(*
Geodetic Ellipsoid
----------------

Overview
================

Represents a geodetic reference ellipsoid (but not a geodetic datum). Contains functions for transitioning between latitude/longitude and XYZ coordinates.

To access standard ellipsoids use the GVL 'GeoEllipsoids'.	They cannot be copied, but you can use REFERENCE TO types to keep a shorthand copy somewhere.

.. note:: When creating an instance of this FB you *must* provide the name, semimajor axis, and flattening due to the use of FB_init parameters.
*)
{attribute 'no_assign'}
FUNCTION_BLOCK GeoEllipsoid
VAR_INPUT
END_VAR
VAR_OUTPUT
END_VAR
VAR
	Name_ : T_MaxString;
	SemiMajorAxis_ : LREAL;
	Flattening_ : LREAL;
END_VAR

METHOD FB_init : BOOL
VAR_INPUT
	bInitRetains : BOOL; // if TRUE, the retain variables are initialized (warm start / cold start)
	bInCopyCode : BOOL;  // if TRUE, the instance afterwards gets moved into the copy code (online change)
	
	eName : T_MaxString;
	eSemiMajorAxis : LREAL;//meters
	eFlattening : LREAL;//very small number
END_VAR
Name_ := eName;
SemiMajorAxis_ := eSemiMajorAxis;
Flattening_ := eFlattening;
END_METHOD

PROPERTY PUBLIC Flattening : LREAL
GET
Flattening := Flattening_;
END_GET
END_PROPERTY

METHOD PUBLIC GetCartesianFromGeodetic : Vector3
VAR_INPUT
	P : GeoPosition;
END_VAR
VAR
	N : LREAL;
END_VAR
N := GetNormalRadiusOfCurvature(P.LatitudeRad);

GetCartesianFromGeodetic.X := (N + P.Elevation) * COS(P.LatitudeRad) * COS(P.LongitudeRad);
GetCartesianFromGeodetic.Y := (N + P.Elevation) * COS(P.LatitudeRad) * SIN(P.LongitudeRad);
GetCartesianFromGeodetic.Z := ((1.0 - GetEccentricitySquared())*N + P.Elevation) * SIN(P.LatitudeRad);
END_METHOD

METHOD PROTECTED GetEccentricitySquared : LREAL
VAR_INPUT
END_VAR
GetEccentricitySquared := (2.0-Flattening)*Flattening;
END_METHOD

METHOD PROTECTED GetGeocentricLatitude : LREAL//radians
VAR_INPUT
	GeodeticLatitude : LREAL;//radians
END_VAR
GetGeocentricLatitude := ATAN((1-Flattening_) * (1-Flattening_)*TAN(GeodeticLatitude));
END_METHOD

METHOD PUBLIC GetGeodeticFromCartesian : GeoPosition
VAR_INPUT
	V : Vector3;
END_VAR
VAR
	RadLatitude_2 : LREAL;// 		'Q^2' 		from paper
	Magnitude_2 : LREAL;// 			'r^2' 		from paper
	Eccentricity_2 : LREAL;// 		'E^2' 		from paper
	AdjustedMag_2 : LREAL;// 		'r^2 - E^2' from paper
	SemiMinorConfocal_2 : LREAL;// 	'u^2' 		from paper
	SemiMajorConfocal_2 : LREAL;// 	'u^2' + E^2 from paper
	TanGeocentricLatitude : LREAL;// tan(beta) 	from paper
	GeocentricLatitude : LREAL;//   'beta' 		from paper
	AxialElevation : LREAL;
	RadialElevation : LREAL;
END_VAR
//stolen from : http://ir.lib.ncku.edu.tw/bitstream/987654321/39750/1/3011200501001.pdf
//error is <1mm for anything within 100km of the surface of the earth

RadLatitude_2 := V.X*V.X + V.Y*V.Y;
Magnitude_2 := RadLatitude_2 + V.Z* V.Z;

//right at pole longitude is indetermiante
IF RadLatitude_2 = 0 THEN
	GetGeodeticFromCartesian.LongitudeRad := 0;
ELSE
	GetGeodeticFromCartesian.LongitudeRad := atan2(V.Y,V.X);//eq 4c from paper
END_IF

//too close to poles for stuff to work well
IF RadLatitude_2 < (SemiMajorAxis * SemiMinorAxis * 1E-32) THEN
	//center of earth...angles dont even matter anymore
	IF V.Z = 0 THEN
		GetGeodeticFromCartesian.LatitudeRad := 0;
		GetGeodeticFromCartesian.Elevation := Magnitude_2;
	ELSE
		GetGeodeticFromCartesian.LatitudeRad := PI /2 * V.Z / ABS(V.Z);
		GetGeodeticFromCartesian.Elevation := ABS(V.Z) - SemiMinorAxis;
	END_IF;
ELSE
	Eccentricity_2 := SemiMajorAxis*SemiMajorAxis - SemiMinorAxis * SemiMinorAxis;
	AdjustedMag_2 := Magnitude_2 - Eccentricity_2;
	SemiMinorConfocal_2 := 0.5*AdjustedMag_2 + 0.5*SQRT(EXPT(AdjustedMag_2,2) + 4*Eccentricity_2*V.Z*V.Z); //eq 4a from paper
	SemiMajorConfocal_2 := SemiMinorConfocal_2 + Eccentricity_2;
	IF SQRT(SemiMinorConfocal_2) / SQRT(SemiMajorConfocal_2) < 10E-10 THEN
		//avoid divide by near zero when confocal is nearly flat and assumption of geocentric latidude equivalence atan(confocal) ~= atan(ellipsoid) stops being true
		IF V.Z = 0 THEN
			GeocentricLatitude := 0;
		ELSE
			GeocentricLatitude := PI/2 * V.Z/ABS(V.Z);
		END_IF;
		GetGeodeticFromCartesian.LatitudeRad := GeocentricLatitude;
	ELSE
		TanGeocentricLatitude := (SQRT(SemiMajorConfocal_2) * V.Z) / (SQRT(SemiMinorConfocal_2)*SQRT(RadLatitude_2));
		GeocentricLatitude := ATAN(TanGeocentricLatitude); //eq 6 from paper
		GetGeodeticFromCartesian.LatitudeRad := ATAN(SemiMajorAxis / SemiMinorAxis * TanGeocentricLatitude);
	END_IF;
	
	AxialElevation := V.Z - SemiMinorAxis*SIN(GeocentricLatitude);
	RadialElevation := SQRT(RadLatitude_2) - SemiMajorAxis*COS(GeocentricLatitude);
	
	GetGeodeticFromCartesian.Elevation := SQRT(AxialElevation*AxialElevation + RadialElevation*RadialElevation); //eq 7 from paper
	IF AxialElevation < 0 AND RadialElevation < 0 THEN
		GetGeodeticFromCartesian.Elevation := -1 * GetGeodeticFromCartesian.Elevation;
	END_IF

END_IF
END_METHOD

METHOD PROTECTED GetNormalRadiusOfCurvature : LREAL
VAR_INPUT
	lat : LREAL;//radians
END_VAR
VAR
	acosf : LREAL;
	bcosf : LREAL;
	den : LREAL;
END_VAR
acosf := SemiMajorAxis * COS(lat);
bcosf := GetSemiMinorAxis() * SIN(lat);
den := SQRT(acosf*acosf + bcosf*bcosf);
IF den = 0 THEN
	GetNormalRadiusOfCurvature := 0;
	ADSLOGSTR(ADSLOG_MSGTYPE_WARN,'GeodeticPosition::GetNormalRadiusOfCurvature Divide By Zero attempt in reference ellipsoid %s',Name);
	RETURN;
END_IF
GetNormalRadiusOfCurvature := SemiMajorAxis*SemiMajorAxis/den;
END_METHOD

METHOD PROTECTED GetSemiMinorAxis : LREAL
VAR_INPUT
END_VAR
GetSemiMinorAxis := SemiMajorAxis * (1-Flattening);
END_METHOD

METHOD PUBLIC GetTangentEnuRotation : RMatrix
VAR_INPUT
	P : GeoPosition;
END_VAR
VAR
	R_ENU : RMatrix;
	R_Lon : Rmatrix;
	R_Lat : Rmatrix;
	V : Vector3;
END_VAR
GetTangentEnuRotation := GetTangentXyuRotation(P,0.0);
RETURN;

//ECEF has X as 'up',   y as 'east',  Z as 'north' as lat=lon=0, translated to surface
//ENU  has X as 'east', y as 'north', z as 'up'
//therefore, the base rotation (ignoring lat/lon changes) should be: (projecting ENU unit vecotrs onto ECEF CS)
// [  0   0   1
//    1   0   0
//    0   1   0   ]

GetTangentEnuRotation.FillTrapezoidal(0,0,0);
GetTangentEnuRotation.SetRC(1,0,1);
GetTangentEnuRotation.SetRC(2,1,1);
GetTangentEnuRotation.SetRC(0,2,1);


R_Lon.SetFromAngle(P.LongitudeRad,Dimension.Z);//positive intrinsic rotation around ECEF Z
R_Lat.SetFromAngle(-1*P.LatitudeRad,Dimension.Y);//negative instrinsic rotation around rotated ECEF Y

GetTangentEnuRotation.RotateBy(R_Lat);
GetTangentEnuRotation.RotateBy(R_Lon);
END_METHOD

METHOD PUBLIC GetTangentEnuTransform : HMatrix
VAR_INPUT
	P : GeoPosition;
END_VAR
VAR
	R_ENU : RMatrix;
	R_Lon : Rmatrix;
	R_Lat : Rmatrix;
	V : Vector3;
END_VAR
V := GetCartesianFromGeodetic(P);
GetTangentEnuTransform.SetFromComponents(GetTangentEnuRotation(P),V);
END_METHOD

METHOD PUBLIC GetTangentXyuRotation : RMatrix
VAR_INPUT
	P : GeoPosition;
	Angle : LREAL;//radians of extra angle around the 'up' vector, from ENU
END_VAR
VAR
	R_ENU : RMatrix;
	R_Lon : Rmatrix;
	R_Lat : Rmatrix;
	RHeading : RMatrix;
	V : Vector3;
END_VAR
//ECEF has X as 'up',   y as 'east',  Z as 'north' as lat=lon=0, translated to surface
//ENU  has X as 'east', y as 'north', z as 'up'
//therefore, the base rotation (ignoring lat/lon changes) should be: (projecting ENU unit vecotrs onto ECEF CS)
// [  0   0   1
//    1   0   0
//    0   1   0   ]

GetTangentXyuRotation.SetFromAngle(Angle,Dimension.Z);

R_ENU.FillTrapezoidal(0,0,0);
R_ENU.SetRC(1,0,1);
R_ENU.SetRC(2,1,1);
R_ENU.SetRC(0,2,1);

R_Lon.SetFromAngle(P.LongitudeRad,Dimension.Z);//positive intrinsic rotation around ECEF Z
R_Lat.SetFromAngle(-1*P.LatitudeRad,Dimension.Y);//negative instrinsic rotation around rotated ECEF Y

GetTangentXyuRotation.RotateBy(R_ENU);
GetTangentXyuRotation.RotateBy(R_Lat);
GetTangentXyuRotation.RotateBy(R_Lon);
END_METHOD

METHOD PUBLIC GetTangentXyuTransform : HMatrix
VAR_INPUT
	P : GeoPosition;
	Angle : LREAL;//radians of extra normal rotation
END_VAR
VAR
	R_ENU : RMatrix;
	R_Lon : Rmatrix;
	R_Lat : Rmatrix;
	V : Vector3;
END_VAR
V := GetCartesianFromGeodetic(P);
GetTangentXyuTransform.SetFromComponents(GetTangentXyuRotation(P,Angle),V);
END_METHOD

PROPERTY PUBLIC Name : T_MaxString
GET
Name := Name_;
END_GET
END_PROPERTY

//meters
PROPERTY PUBLIC SemiMajorAxis : LREAL
GET
SemiMajorAxis := SemiMajorAxis_;
END_GET
END_PROPERTY

PROPERTY PUBLIC SemiMinorAxis : LREAL
GET
SemiMinorAxis := SemiMajorAxis*(1-Flattening);
END_GET
END_PROPERTY

END_FUNCTION_BLOCK

(* stored: Version 1.1.0.1, ProductVersion 3.1.4024.9
   POU GeoEllipsoid: Id {5fa9ec91-c8df-4619-93de-f428fe8da353}, SpecialFunc None
   Folder Helpers: Id {b81f80d4-2bbb-4268-8ddd-c7326c54d401}
   Folder Properties: Id {b4f92432-ea7a-4ff4-815d-4808dee4ca34}
   Folder Protected: Id {d95a2200-fe2b-4706-b87d-15a39d09296c}
   Method FB_init: Id {356473b9-f5c8-4741-9e86-0658e3600f83}
   Property Flattening: Id {34b2fe7f-e49d-4b2c-8e6e-38d008c42ac1}
   Get Get: Id {5861998b-a1c7-428b-b4da-036da0771533}
   Method GetCartesianFromGeodetic: Id {3dee90e0-402c-4ec5-8ec8-6eb06ee928ca}
   Method GetEccentricitySquared: Id {dcf07e5e-00c3-480f-9648-fb9fcd18870b}
   Method GetGeocentricLatitude: Id {7fa6146d-71cd-4c31-88c4-e5b241b37441}
   Method GetGeodeticFromCartesian: Id {9f899f33-9489-4cc0-a19d-4c589c0cda4f}
   Method GetNormalRadiusOfCurvature: Id {1cc8408c-a28c-42ab-bd8d-21272b17e8e7}
   Method GetSemiMinorAxis: Id {10667ac4-3728-46cd-b99e-93e77afe5ab6}
   Method GetTangentEnuRotation: Id {990d09c8-060e-47ac-a561-59f9dceba14c}
   Method GetTangentEnuTransform: Id {a5892b07-6af9-48fe-b43a-dae14b491220}
   Method GetTangentXyuRotation: Id {083e21a0-e6de-41d9-9dcb-5bd7a8d96a35}
   Method GetTangentXyuTransform: Id {1e75e771-e680-4e4e-876e-379512ece41b}
   Property Name: Id {11b38d1a-0e13-4252-824e-6e3d0a3d3677}
   Get Get: Id {dcb313e4-5062-49e4-b4c0-aa22e54019b5}
   Property SemiMajorAxis: Id {a8d72ca4-bbbb-4088-a6eb-591ebbd96221}
   Get Get: Id {7f8fad21-a403-4c2d-bed6-8bb7db93b188}
   Property SemiMinorAxis: Id {c6aadc78-4572-4d9c-8819-d08f87b272c4}
   Get Get: Id {8345bad9-ea91-4c40-9211-991e6f818527} *)
